(*
SPDX-FileCopyrightText: © 2026 Oleksandr Tiutyk <trofimich@gmail.com>
SPDX-License-Identifier: MIT
License: https://opensource.org/license/mit
*)

(*!
<summary>Reports a field or property value outside the range accepted by the caller.</summary>
<description>
The caller detects the member error; Throw records diagnostics rather than inspecting the object. Dynamic
instances and clones belong to the current task memory manager until cleanup. Value text is limited to 255
characters. Longer STRING and WSTRING inputs use a 254-character prefix followed by an ellipsis.
</description>
*)
INTERFACE IDataMemberOutOfRangeException EXTENDS IGeneralException

(*!
<summary>Formats the rejected member and propagates the exception.</summary>
<description>
Call in the owning cyclic task, not during FB_init. Builds a member diagnostic and captures source and
timestamps with zero error code and no inner cause. Input storage is not retained. Allocation failure uses the
shared terminal memory mechanism. Uses the shared ANY formatter; STRING and WSTRING values longer than 255
characters retain their first 254 characters followed by an ellipsis. Exactly 255 characters remain unchanged.
</description>
<param name="dataMemberName">Name of the field or property rejected by the caller.</param>
<param name="dataMemberValue">Live value to describe; string inputs must be null-terminated.</param>
*)
METHOD Throw
VAR_INPUT
	sourceNamespaceName : STRING;
	sourceClassName : STRING;
	sourcePOUName : STRING;
	sourcePosition : STRING;
	dataMemberName : STRING;
	dataMemberValue : ANY;
END_VAR
END_METHOD

END_INTERFACE

(* stored: Version 1.1.0.1
   Itf IDataMemberOutOfRangeException: Id {cf663f39-5e05-4307-91b0-0444aac88c2e}
   Method Throw: Id {c468a2b6-6032-48d2-a9d4-533017cb99d6} *)
